{attribute 'hide_all_locals'}
{attribute 'conditionalshow'}
FUNCTION_BLOCK FB_NumberOfDevice
VAR_INPUT
	{attribute 'hide'}
	diActualNumberOfDevices			: DINT;							//Actual Number for this Device
	{attribute 'hide'}
	diMaxNumberOfDevices			: DINT;							//Max Numbers for this Device
	{attribute 'hide'}
	udiCounterOnlineChange			: UDINT;						//Actual Counter for Online change
END_VAR
VAR_OUTPUT
	{attribute 'hide'}
	bNumberIsCalculatet				: BOOL;							//Number for this Device ic calculatet
	{attribute 'hide'}
	bFPNumberIsCalculatet			: BOOL;							//Number for this Device ic calculatet. Only positive Edge
	{attribute 'hide'}
	bOnlineChange					: BOOL;							//Its true for 1 cycle when a Online change was success
	{attribute 'hide'}
	diNumberForThisDevice			: DINT;							//Number for this Device
	{attribute 'hide'}
	diNumberOfTotalDevices			: DINT;							//Total Devices without Limits
END_VAR
VAR
	FPCalculatet					: R_TRIG;						//Internal positive edge
	udiCounterOnlineChange_CP		: UDINT;						//Counter online changen to compare with the original input variable
END_VAR

//Creator : Kai Ebensperger
//Company : Lynus AG
//Date : 29.05.2021
//Version : 1.0.0.0

//With this Function its possible to count a number for a Device in PLC
//The number reset and renew when we have a online change on the plc

//Calculate the number of Device
IF NOT bNumberIsCalculatet THEN
	IF diActualNumberOfDevices < diMaxNumberOfDevices THEN diNumberForThisDevice := diActualNumberOfDevices + 1; bNumberIsCalculatet := TRUE; END_IF 
		diNumberOfTotalDevices := diActualNumberOfDevices + 1;
			FPCalculatet.CLK := TRUE;
				diNumberForThisDevice := LIMIT(0,diNumberForThisDevice,diMaxNumberOfDevices);		
END_IF 
	//Reset when we have a online change
	IF bOnlineChange THEN bOnlineChange := FALSE; END_IF
		IF udiCounterOnlineChange <> udiCounterOnlineChange_CP THEN
			bNumberIsCalculatet := FALSE;
				diNumberForThisDevice := 0;
					diNumberOfTotalDevices := diNumberForThisDevice;
						udiCounterOnlineChange_CP := udiCounterOnlineChange;   
							bOnlineChange := TRUE;	
								FPCalculatet.CLK := FALSE;			
		END_IF  
		
FPCalculatet(CLK:= , Q=> bFPNumberIsCalculatet);

END_FUNCTION_BLOCK

(* stored: Version 1.1.0.1, ProductVersion 3.1.4024.6
   POU FB_NumberOfDevice: Id {5a6b7445-7e7f-4b94-bc14-8ae5366a360f}, SpecialFunc None *)
